// TIA Portal V20 export
TYPE "LKinCtrl_PointEditor_typePointConfigurationInternalEvents"
// stored: Access Published
   STRUCT
      selectionChanged { ExternalAccessible := 'False'; ExternalVisible := 'False'; ExternalWritable := 'False'} : Struct
         trigger : Bool;   // triggers event. Only true for 1 cycle.
         noSelection : Bool;
         selectedIndex : DInt;
      END_STRUCT;
      touchUp { ExternalAccessible := 'False'; ExternalVisible := 'False'; ExternalWritable := 'False'} : Struct
         trigger : Bool;
         index : DInt := -1;   // Index in point table. -1: currently selected point
         keepName : Bool := TRUE;   // Ignores the new name.
         point : "LKinCtrl_typePoint";   // New point.
      END_STRUCT;
   END_STRUCT;
END_TYPE
